RoboDK station: New Station (1).rdk

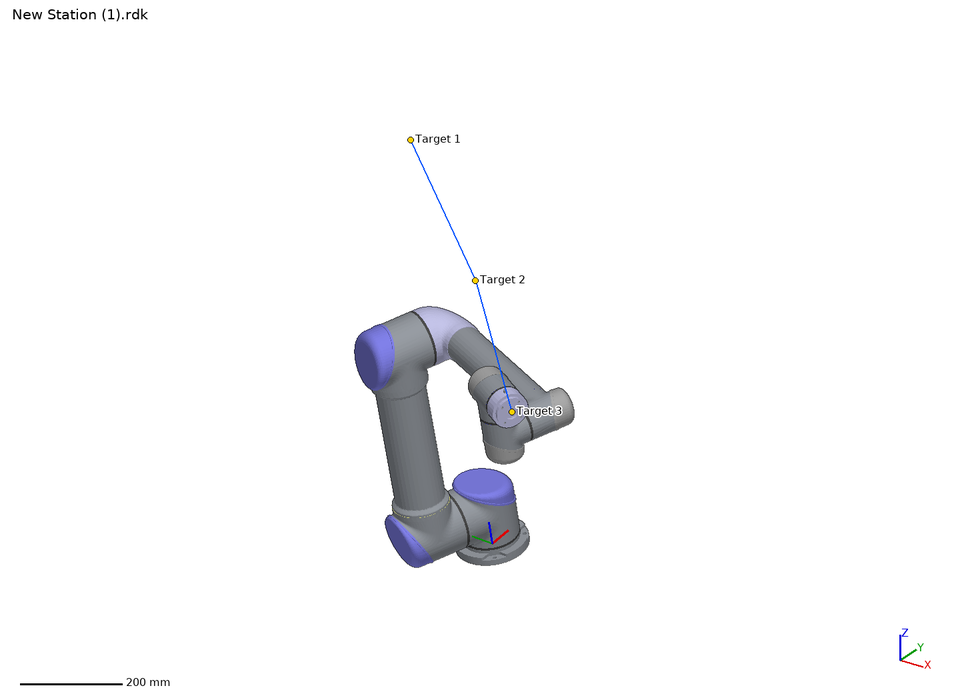
[picture v0: the station drawn from its stored meshes, robots at their saved joint values, targets as dots, program paths as lines]
Station New Station (1). Poses are relative to the parent item; angles as X-Y-Z fixed-axis rotations.
  - frame UR5 Base at (-2.33, -26.72, -68.15) mm, rotated rx 0 ry -11.49 rz 85.03 deg
    - robot UR5: 6 axes, payload 5 kg, reach 850 mm, repeatability 0.1 mm, weight 18.4 kg
        modified DH rows (alpha deg, a mm, theta deg, d mm): 0, 0, 0, 89.2; 90, 0, 180, 0; 0, 425, 0, 0; 0, 392.43, 0, 109; -90, 0, 0, 93.65; 90, 0, 180, 82
        joint limits [-360, -360, -360, -360, -360, -360] to [360, 360, 360, 360, 360, 360]; home [0, -90, -90, 0, 90, 0]; saved at [-111.41, -87.13, -91.72, 0, 84.84, 0]
    - target Target 1 (Cartesian target) at (-89.32, -38.16, 1039.51) mm, rotated rx -89.99 ry 0 rz 153.43 deg; joints [-138.478, -78.294, -9.305, -92.39, 111.908, 0.005] of UR5
    - target Target 2 (Cartesian target) at (-231.21, -293.78, 877.75) mm, rotated rx -64.33 ry 2.24 rz 153.94 deg; joints [-109.716, -91.987, -49.562, -12.614, 83.315, -0.741] of UR5
    - target Target 3 (Cartesian target) at (-272.92, -377.25, 616.81) mm, rotated rx -88.85 ry 0.1 rz 153.43 deg; joints [-111.41, -87.13, -91.72, 0, 84.84, 0] of UR5
    - target Target 4 (Cartesian target) at (-272.92, -377.25, 616.81) mm, rotated rx -88.85 ry 0.1 rz 153.43 deg; joints [-111.41, -87.13, -91.72, 0, 84.84, 0] of UR5
  - program Prog1 (5 instructions, listed below)
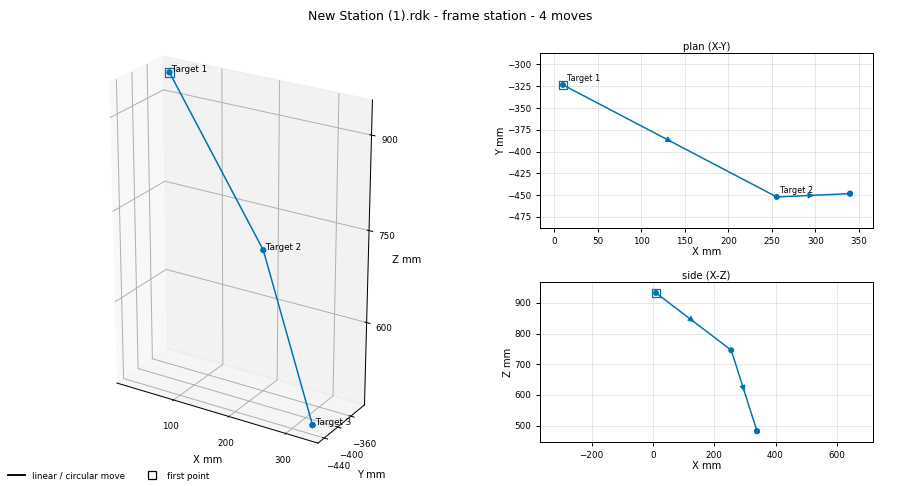
[picture p0: tool path of New Station (1).rdk in frame station, 4 of 4 moves have a stored position in this frame; points joined in program order, loops and branches not executed]

--- program Prog1 (robot UR5) ---
  Set Ref.: UR5 Base
  MoveL (Target 1)
  MoveL (Target 2)
  MoveL (Target 3)
  MoveL (Target 4)
